// TwinCAT 3 PLC project Robot_lib
// Title: UR3e_Robot
// Company: Thomas More
// Author: Arno Joosen
// ProjectVersion: 1.0.0
// ProgramVersion: 3.1.4023.0
// libraries:
//   Tc2_Standard, * (Beckhoff Automation GmbH)
//   Tc2_System, * (Beckhoff Automation GmbH)
//   Tc3_Module, * (Beckhoff Automation GmbH)
// project tree:
//   DUTs/Converut Unions/ BitStruct_Byte.TcDUT, ByteStruct.TcDUT, INT_ByteArray.TcDUT, REAL_ByteArray.TcDUT
//   DUTs/ Robot_Error.TcDUT, UR3e_Robot.TcDUT
//   / PlcTask.TcTTO
//   POUs/GetValue/ Robot_Get_Bool.TcPOU, Robot_Get_Int.TcPOU, Robot_Get_Real.TcPOU
//   POUs/ Robot_Start_Job.TcPOU, Robot_Update.TcPOU
//   POUs/SetValue/ Robot_Set_Bool.TcPOU, Robot_Set_Int.TcPOU, Robot_Set_Real.TcPOU
//   SubFuncites/ Robot_Chek_errors.TcPOU
// (motion and I/O tree: see PLC project rfid_lib)
// real-time tasks:
//   TASK PlcTask: cycle T#10ms, priority 20, ADS port 350
//   TASK PlcTask1: cycle T#10ms, priority 21, ADS port 351
//   TASK PlcTask2: cycle T#10ms, priority 22, ADS port 352
//   TASK PlcTask3: cycle T#10ms, priority 23, ADS port 353

CONFIGURATION Robot_lib
    RESOURCE PLC ON TwinCAT3
        TASK PlcTask(INTERVAL := T#10ms, PRIORITY := 22);
        PROGRAM MAIN WITH PlcTask : MAIN;
    END_RESOURCE
END_CONFIGURATION

// ---- DUTs/Converut Unions/BitStruct_Byte.TcDUT
TYPE BitStruct_Byte :
UNION
	Value : BYTE;
	SValue : ByteStruct;
END_UNION
END_TYPE

// ---- DUTs/Converut Unions/ByteStruct.TcDUT
TYPE ByteStruct :
STRUCT
	Bit0 : BIT;
	Bit1 : BIT;
	Bit2 : BIT;
	Bit3 : BIT;
	Bit4 : BIT;
	Bit5 : BIT;
	Bit6 : BIT;
	Bit7 : BIT;
END_STRUCT
END_TYPE

// ---- DUTs/Converut Unions/INT_ByteArray.TcDUT
TYPE INT_ByteArray :
UNION
	AValue : ARRAY[0..4] OF BYTE;
	Value : DINT;
END_UNION
END_TYPE

// ---- DUTs/Converut Unions/REAL_ByteArray.TcDUT
TYPE REAL_ByteArray :
UNION
	AValue : ARRAY[0..4] OF BYTE;
	Value : REAL;
END_UNION
END_TYPE

// ---- DUTs/Robot_Error.TcDUT
{attribute 'qualified_only'}
{attribute 'strict'}
TYPE Robot_Error :
(
	None := 0,
	Not_Power_On := 1,
	Not_Running := 2,
	Protective_Stopped := 3,
	Safeguard_Stopped := 4,
	System_Emergency_Stopped := 5,
	Robot_Emergency_Stopped := 6,
	Emergency_Stopped := 7,
	Stopped_Due_To_Safety := 8,
	Profinet := 9
) UINT;
END_TYPE

// ---- DUTs/UR3e_Robot.TcDUT
TYPE UR3e_Robot :
STRUCT
	// input
	PnioBoxState AT %I* : UINT;
		//0 = No error
		//1 = Profinet device state machine is in boot mode
		//2 = Device not found
		//3 = The stationname is not unique
		//4 = IP could not be set
		//5 = IP conflict
		//6 = DCP set was not successful
		//7 = Watchdog error
		//8 = Datahold error
		//9 = RTC3: Sync mode could not be initiated
		//10 = Profinet controller has a link error
		//11 = The aliasname is not unique
		//12 = The automatic name assignement isn't possible - wrong device type
		//13 = IOC-AR is established but no application ready
		//14 = IOC-AR is established but module difference
		//15 = At least one InputCR is invalid, provider in stop or problemindicator is set
		//16 = At least one OutputCR is invalid, provider in stop or problemindicator is set
		//31 = Only for EtherCAT gateways: WC-State of cyclic EtherCAT frame is 1
	RobotState_And_Safety AT %I* : ARRAY[0..31] OF BYTE;
	GPR_BIT AT %I* : ARRAY[0..7] OF BYTE;
	GPR_INT AT %I* : ARRAY[0..95] OF BYTE;
	GPR_REAL AT %I* : ARRAY[0..95] OF BYTE;

	// ouput
	GPR1 AT %Q* : ARRAY[0..99] OF BYTE;
	GPR2 AT %Q* : ARRAY[0..99] OF BYTE;
END_STRUCT
END_TYPE

// ---- POUs/GetValue/Robot_Get_Bool.TcPOU
FUNCTION Robot_Get_Bool : BOOL
VAR_INPUT
	Num : UINT;
END_VAR
VAR_IN_OUT
	Robot : UR3e_Robot;
	Value : BOOL;
END_VAR
VAR
	Row : UINT;
	Colom : UINT;
	BitArray : BitStruct_Byte;
END_VAR

IF Num <= 63 AND (NOT (Num = 0)) THEN
	Row := Num/8;
	Colom := Num MOD 8;
	BitArray.Value := Robot.GPR_BIT[Row];
	CASE Colom OF
		0:
			Value := BitArray.SValue.Bit0;
		1:
			Value := BitArray.SValue.Bit1;
		2:
			Value := BitArray.SValue.Bit2;		
		3:
			Value := BitArray.SValue.Bit3;
		4:
			Value := BitArray.SValue.Bit4;
		5:
			Value := BitArray.SValue.Bit5;
		6:
			Value := BitArray.SValue.Bit6;
		7:
			Value := BitArray.SValue.Bit7;
	END_CASE
	Robot_Get_Bool := TRUE;
ELSE
	Robot_Get_Bool := FALSE;
END_IF

END_FUNCTION

// ---- POUs/GetValue/Robot_Get_Int.TcPOU
FUNCTION Robot_Get_Int : BOOL
VAR_INPUT
	Num : UINT;
END_VAR
VAR_IN_OUT
	Robot : UR3e_Robot;
	Value : DINT;
END_VAR
VAR
	Row : UINT;
	INTArray : INT_ByteArray;
	i : UINT;
END_VAR

IF Num <= 23 THEN
	Row := Num * 4;
	FOR i:=0 TO 3 BY 1 DO
		INTArray.AValue[3-i] := Robot.GPR_INT[Row+i];
	END_FOR
	
	Value := INTArray.Value;
	Robot_Get_Int := TRUE;
ELSE
	Robot_Get_Int := FALSE;
END_IF

END_FUNCTION

// ---- POUs/GetValue/Robot_Get_Real.TcPOU
FUNCTION Robot_Get_Real : BOOL
VAR_INPUT
	Num : UINT;
END_VAR
VAR_IN_OUT
	Robot : UR3e_Robot;
	Value : REAL;
END_VAR
VAR
	Row : UINT;
	REALArray : REAL_ByteArray;
	i : UINT;
END_VAR

IF Num <= 23 THEN
	Row := Num * 4;
	FOR i:=0 TO 3 BY 1 DO
		REALArray.AValue[3-i] := Robot.GPR_REAL[Row+i];
	END_FOR
	
	Value := REALArray.Value;
	Robot_Get_Int := TRUE;
ELSE
	Robot_Get_Int := FALSE;
END_IF

END_FUNCTION

// ---- POUs/Robot_Start_Job.TcPOU
FUNCTION Robot_Start_Job : Robot_Error
VAR_INPUT
	JobID : UDINT;
END_VAR
VAR_IN_OUT
	Robot : UR3e_Robot;
END_VAR
VAR
	bitArray : BitStruct_Byte;
	IntArray : INT_ByteArray;
	i : UINT;
END_VAR

Robot_Start_Job := Robot_Chek_errors(Robot:= Robot);

IF Robot_Start_Job = Robot_Error.None AND (NOT((Robot.GPR_BIT[0] AND 2#00000001) = 2#00000001)) THEN
	
	// zet job is in int0
	IntArray.Value := JobID;
	FOR i := 0 TO 3 BY 1 DO
		Robot.GPR1[4+i] := IntArray.AValue[3-i];
	END_FOR
	
	// zet bool0 true
	bitArray.Value := Robot.GPR1[0];
	bitArray.SValue.Bit0 := TRUE;
	Robot.GPR1[0] := bitArray.Value;
END_IF

END_FUNCTION

// ---- SubFuncites/Robot_Chek_errors.TcPOU
FUNCTION Robot_Chek_errors : Robot_Error
VAR_INPUT
	Robot : UR3e_Robot;
END_VAR
VAR
END_VAR

IF NOT((Robot.RobotState_And_Safety[16] AND 2#00000001) = 2#00000001) THEN // Not Power On
	Robot_Chek_errors := Robot_Error.Not_Power_On;
ELSIF NOT ((Robot.RobotState_And_Safety[16] AND 2#00000010) = 2#00000010) THEN // Not Running
	Robot_Chek_errors := Robot_Error.Not_Running;
ELSIF (Robot.RobotState_And_Safety[28] AND 2#00000100) = 2#00000100 THEN // Protective Stopped
	Robot_Chek_errors := Robot_Error.Protective_Stopped;
ELSIF (Robot.RobotState_And_Safety[28] AND 2#00010000) = 2#00010000 THEN // Safeguard Stopped
	Robot_Chek_errors := Robot_Error.Safeguard_Stopped;
ELSIF (Robot.RobotState_And_Safety[28] AND 2#00100000) = 2#00100000 THEN // System Emergency Stopped
	Robot_Chek_errors := Robot_Error.System_Emergency_Stopped;
ELSIF (Robot.RobotState_And_Safety[28] AND 2#01000000) = 2#01000000 THEN // Robot Emergency Stopped
	Robot_Chek_errors := Robot_Error.Robot_Emergency_Stopped;
ELSIF (Robot.RobotState_And_Safety[28] AND 2#10000000) = 2#10000000 THEN // Emergency Stopped
	Robot_Chek_errors := Robot_Error.Emergency_Stopped;
ELSIF (Robot.RobotState_And_Safety[29] AND 2#00000100) = 2#00000100 THEN // Stopped Due To Safety
	Robot_Chek_errors := Robot_Error.Stopped_Due_To_Safety;
ELSIF NOT(Robot.PnioBoxState = 0) THEN // profinet error
	Robot_Chek_errors := Robot_Error.Profinet;
ELSE
	Robot_Chek_errors := Robot_Error.None;
END_IF

END_FUNCTION

// ---- POUs/Robot_Update.TcPOU
FUNCTION_BLOCK Robot_Update
VAR_INPUT
END_VAR
VAR_OUTPUT
	Free : BOOL;
	Error : Robot_Error;
END_VAR
VAR_IN_OUT
	Robot : UR3e_Robot;
END_VAR
VAR
	bitArray : BitStruct_Byte;
END_VAR

Error := Robot_Chek_errors(Robot:= Robot);

// chek of robot bezig is
IF (Robot.GPR_BIT[0] AND 2#00000001) = 2#00000001 THEN
	// zet run varibel FALSE zo dat robot de job niet bleift heralen
	bitArray.Value := Robot.GPR1[0];
	bitArray.SValue.Bit0 := FALSE;
	Robot.GPR1[0] := bitArray.Value;
	Free := FALSE;
ELSE
	Free := TRUE;
END_IF

END_FUNCTION_BLOCK

// ---- POUs/SetValue/Robot_Set_Bool.TcPOU
FUNCTION Robot_Set_Bool : BOOL
VAR_INPUT
	Num : UINT;
	Value : BOOL;
END_VAR
VAR_IN_OUT
	Robot : UR3e_Robot;
END_VAR
VAR
	Row : UINT;
	Colom : UINT;
	BitArray : BitStruct_Byte;
END_VAR

IF Num = 0 OR Num > 63 THEN
	Robot_Set_Int := FALSE;
	RETURN;
END_IF

IF Num < 32 THEN
	Row := Num / 8; // bereken de index in de buffer
	Colom := Num MOD 8; // berken de bit nummer in de byte
	BitArray.Value := RObot.GPR1[Row];
	CASE Colom OF
		0:
			BitArray.SValue.Bit0  := Value;
		1:
			BitArray.SValue.Bit1  := Value;
		2:
			BitArray.SValue.Bit2  := Value;		
		3:
			BitArray.SValue.Bit3  := Value;
		4:
			BitArray.SValue.Bit4  := Value;
		5:
			BitArray.SValue.Bit5  := Value;
		6:
			BitArray.SValue.Bit6  := Value;
		7:
			BitArray.SValue.Bit7  := Value;
	END_CASE
	RObot.GPR1[Row] := BitArray.Value;
	Robot_Set_Int := TRUE;
	RETURN;
	
ELSIF Num > 31 THEN
	Row := (Num-32) / 8; // bereken de index in de buffer
	Colom := (Num-32) MOD 8; // berken de bit nummer in de byte
	BitArray.Value := RObot.GPR2[Row];
	CASE Colom OF
		0:
			BitArray.SValue.Bit0  := Value;
		1:
			BitArray.SValue.Bit1  := Value;
		2:
			BitArray.SValue.Bit2  := Value;		
		3:
			BitArray.SValue.Bit3  := Value;
		4:
			BitArray.SValue.Bit4  := Value;
		5:
			BitArray.SValue.Bit5  := Value;
		6:
			BitArray.SValue.Bit6  := Value;
		7:
			BitArray.SValue.Bit7  := Value;
	END_CASE
	RObot.GPR2[Row] := BitArray.Value;
	Robot_Set_Int := TRUE;
	RETURN;
	
END_IF

END_FUNCTION

// ---- POUs/SetValue/Robot_Set_Int.TcPOU
FUNCTION Robot_Set_Int : BOOL
VAR_INPUT
	Num : UINT;
	Value : DINT;
END_VAR
VAR_IN_OUT
	Robot : UR3e_Robot;
END_VAR
VAR
	Row : UINT;
	INTArray : INT_ByteArray;
	i : UINT;
END_VAR

IF Num = 0 OR Num > 23 THEN
	Robot_Set_Int := FALSE;
	RETURN;
END_IF

IF Num < 12 THEN
	INTArray.Value := Value;
	Row := (Num * 4) + 4; // bereken start byte in buffer
	FOR i:=0 TO 3 BY 1 DO // copy data
		Robot.GPR1[Row+i] := INTArray.AValue[3-i];
	END_FOR
	Robot_Set_Int := TRUE;
	RETURN;
ELSIF Num > 11 THEN
	INTArray.Value := Value;
	Row := ((Num - 12) * 4) + 4; // bereken start byte in buffer
	FOR i:=0 TO 3 BY 1 DO // copy data
		Robot.GPR2[Row+i] := INTArray.AValue[3-i];
	END_FOR
	Robot_Set_Int := TRUE;
	RETURN;
END_IF

END_FUNCTION

// ---- POUs/SetValue/Robot_Set_Real.TcPOU
FUNCTION Robot_Set_Real : BOOL
VAR_INPUT
	Num : UINT;
	Value : REAL;
END_VAR
VAR_IN_OUT
	Robot : UR3e_Robot;
END_VAR
VAR
	Row : UINT;
	REALArray : REAL_ByteArray;
	i : UINT;
END_VAR

IF Num > 23 THEN
	Robot_Set_Int := FALSE;
	RETURN;
END_IF

IF Num < 12 THEN
	REALArray.Value := Value;
	Row := (Num * 4)+52; // bereken start byte in buffer
	FOR i:=0 TO 3 BY 1 DO // copy data
		Robot.GPR1[Row+i] := REALArray.AValue[3-i];
	END_FOR
	Robot_Set_Int := TRUE;
	RETURN;
ELSIF Num > 11 THEN
	REALArray.Value := Value;
	Row := ((Num - 12) * 4) + 52; // bereken start byte in buffer
	FOR i:=0 TO 3 BY 1 DO // copy data
		Robot.GPR2[Row+i] := REALArray.AValue[3-i];
	END_FOR
	Robot_Set_Int := TRUE;
	RETURN;
END_IF

END_FUNCTION
